(*

short summary
=================
This class provides assert statements for unsigned integers  (``UINT``)
It implements the interface :ref:`IUintAssertions`

.. <legal notes>

legal notes
=================
| SPDX-FileCopyrightText: © 2022 ekvip automation GmbH <info@ekvip.de>
| SPDX-License-Identifier: Apache-2.0
| For details check: Apache-2.0_

.. _Apache-2.0: https://www.apache.org/licenses/LICENSE-2.0

.. </legal notes>

methods and properties
=======================

*)

{attribute 'reflection'}
FUNCTION_BLOCK INTERNAL UintAssertions EXTENDS AbstactAssertion IMPLEMENTS IUintAssertions
VAR
END_VAR

(*

short summary
=================
This abstract property returns the class name of the concrete object, 
It's for debugging purpose

.. <legal notes>

legal notes
=================
| SPDX-FileCopyrightText: © 2022 ekvip automation GmbH <info@ekvip.de>
| SPDX-License-Identifier: Apache-2.0
| For details check: Apache-2.0_

.. _Apache-2.0: https://www.apache.org/licenses/LICENSE-2.0

.. </legal notes>

*)

PROPERTY className :CNM_AbstractObject.ClassName
GET
className := 'CNM_AssertionInterfaceLib.UintAssertions';
END_GET
END_PROPERTY

(*

short summary
=================
This assertion method checks if the current value is equal to the expected value

.. <legal notes>

legal notes
=================
| SPDX-FileCopyrightText: © 2022 ekvip automation GmbH <info@ekvip.de>
| SPDX-License-Identifier: Apache-2.0
| For details check: Apache-2.0_

.. _Apache-2.0: https://www.apache.org/licenses/LICENSE-2.0

.. </legal notes>

parameters
=================

*)

METHOD valueIsEqualTo
VAR_INPUT
	(* current value to check *)
	currentValue	:UINT;
	(* expected value to compare *)
	expectedValue	:UINT;
	(* message if the assertion is false *)
	message			:AssertMessage;
END_VAR
IF (currentValue <> expectedValue) THEN
	THIS^.assertionWasWrong(message, THIS^.getDebugInfo('valueIsEqualTo'));
END_IF
END_METHOD

(*

short summary
=================
This assertion method checks if the current value is even

.. <legal notes>

legal notes
=================
| SPDX-FileCopyrightText: © 2022 ekvip automation GmbH <info@ekvip.de>
| SPDX-License-Identifier: Apache-2.0
| For details check: Apache-2.0_

.. _Apache-2.0: https://www.apache.org/licenses/LICENSE-2.0

.. </legal notes>

parameters
=================

*)

METHOD valueIsEven
VAR_INPUT
	(* current value to check *)
	currentValue	:UINT;
	(* message if the assertion is false *)
	message			:Tc2_System.T_MaxString;
END_VAR
IF ((currentValue MOD 2) <> 0) THEN
	THIS^.assertionWasWrong(message, THIS^.getDebugInfo('valueIsEven'));
END_IF
END_METHOD

(*

short summary
=================
This assertion method checks if the current value is greater than the less value

.. <legal notes>

legal notes
=================
| SPDX-FileCopyrightText: © 2022 ekvip automation GmbH <info@ekvip.de>
| SPDX-License-Identifier: Apache-2.0
| For details check: Apache-2.0_

.. _Apache-2.0: https://www.apache.org/licenses/LICENSE-2.0

.. </legal notes>

parameters
=================

*)

METHOD valueIsGreaterThan
VAR_INPUT
	(* current value to check *)
	currentValue	:UINT;
	(* less than lower limit *)
	lessValue		:UINT;
	(* message if the assertion is false *)
	message			:AssertMessage;
END_VAR
IF (currentValue <= lessValue) THEN
	THIS^.assertionWasWrong(message, THIS^.getDebugInfo('valueIsGreaterThan'));
END_IF
END_METHOD

(*

short summary
=================
This assertion method checks if the current value is inside a limit

.. attention:: 
	limits are included: ``valueIsInRangeOf(3, 3, 3)`` is a true assertion

.. <legal notes>

legal notes
=================
| SPDX-FileCopyrightText: © 2022 ekvip automation GmbH <info@ekvip.de>
| SPDX-License-Identifier: Apache-2.0
| For details check: Apache-2.0_

.. _Apache-2.0: https://www.apache.org/licenses/LICENSE-2.0

.. </legal notes>

parameters
=================

*)

METHOD valueIsInRangeOf
VAR_INPUT
	(* lower limit for the current value *)
	lowerLimit		:UINT;
	(* current value to check *)
	currentValue	:UINT;
	(* upper limit for the current value *)
	upperLimit		:UINT;
	(* message if the assertion is false *)
	message			:AssertMessage;
END_VAR
IF (
	(currentValue < lowerLimit)
	OR (currentValue > upperLimit)
) THEN
	THIS^.assertionWasWrong(message, THIS^.getDebugInfo('valueIsInRangeOf'));
END_IF
END_METHOD

(*

short summary
=================
This assertion method checks if the current value is less than the greater value

.. <legal notes>

legal notes
=================
| SPDX-FileCopyrightText: © 2022 ekvip automation GmbH <info@ekvip.de>
| SPDX-License-Identifier: Apache-2.0
| For details check: Apache-2.0_

.. _Apache-2.0: https://www.apache.org/licenses/LICENSE-2.0

.. </legal notes>

parameters
=================

*)

METHOD valueIsLessThan
VAR_INPUT
	(* current value to check *)
	currentValue	:UINT;
	(* greater than upper limit *)
	greaterValue	:UINT;
	(* message if the assertion is false *)
	message			:AssertMessage;
END_VAR
IF (currentValue >= greaterValue) THEN
	THIS^.assertionWasWrong(message, THIS^.getDebugInfo('valueIsLessThan'));
END_IF
END_METHOD

(*

short summary
=================
This assertion method checks if the current value is less than or equal to the maximum value

.. <legal notes>

legal notes
=================
| SPDX-FileCopyrightText: © 2022 ekvip automation GmbH <info@ekvip.de>
| SPDX-License-Identifier: Apache-2.0
| For details check: Apache-2.0_

.. _Apache-2.0: https://www.apache.org/licenses/LICENSE-2.0

.. </legal notes>

parameters
=================

*)

METHOD valueIsMax
VAR_INPUT
	(* current value to check *)
	currentValue	:UINT;
	(* upper limit for the current value *)
	maximumValue	:UINT;
	(* message if the assertion is false *)
	message			:AssertMessage;
END_VAR
IF (currentValue > maximumValue) THEN
	THIS^.assertionWasWrong(message, THIS^.getDebugInfo('valueIsMax'));
END_IF
END_METHOD

(*

short summary
=================
This assertion method checks if the current value is greater than or equal to the minimum value

.. <legal notes>

legal notes
=================
| SPDX-FileCopyrightText: © 2022 ekvip automation GmbH <info@ekvip.de>
| SPDX-License-Identifier: Apache-2.0
| For details check: Apache-2.0_

.. _Apache-2.0: https://www.apache.org/licenses/LICENSE-2.0

.. </legal notes>

parameters
=================

*)

METHOD valueIsMin
VAR_INPUT
	(* current value to check *)
	currentValue	:UINT;
	(* lower limit for the current value *)
	minimumValue	:UINT;
	(* message if the assertion is false *)
	message			:AssertMessage;
END_VAR
IF (currentValue < minimumValue) THEN
	THIS^.assertionWasWrong(message, THIS^.getDebugInfo('valueIsMin'));
END_IF
END_METHOD

(*

short summary
=================
This assertion method checks if the current value is not equal to the unexpected value

.. <legal notes>

legal notes
=================
| SPDX-FileCopyrightText: © 2022 ekvip automation GmbH <info@ekvip.de>
| SPDX-License-Identifier: Apache-2.0
| For details check: Apache-2.0_

.. _Apache-2.0: https://www.apache.org/licenses/LICENSE-2.0

.. </legal notes>

parameters
=================

*)

METHOD valueIsNotEqualTo
VAR_INPUT
	(* current value to check *)
	currentValue	:UINT;
	(* unexpected value to compare *)
	unexpectedValue	:UINT;
	(* message if the assertion is false *)
	message			:AssertMessage;
END_VAR
IF (currentValue = unexpectedValue) THEN
	THIS^.assertionWasWrong(message, THIS^.getDebugInfo('valueIsNotEqualTo'));
END_IF
END_METHOD

(*

short summary
=================
This assertion method checks if the current value is odd

.. <legal notes>

legal notes
=================
| SPDX-FileCopyrightText: © 2022 ekvip automation GmbH <info@ekvip.de>
| SPDX-License-Identifier: Apache-2.0
| For details check: Apache-2.0_

.. _Apache-2.0: https://www.apache.org/licenses/LICENSE-2.0

.. </legal notes>

parameters
=================

*)

METHOD valueIsOdd
VAR_INPUT
	(* current value to check *)
	currentValue	:UINT;
	(* message if the assertion is false *)
	message			:AssertMessage;
END_VAR
IF ((currentValue MOD 2) = 0) THEN
	THIS^.assertionWasWrong(message, THIS^.getDebugInfo('valueIsOdd'));
END_IF
END_METHOD

END_FUNCTION_BLOCK

(* stored: Version 1.1.0.1, ProductVersion 3.1.4024.11
   POU UintAssertions: Id {84cb69cf-f417-49b9-b9fb-83ea1eacb025}, SpecialFunc None
   Property className: Id {717aea52-1536-4993-b7ba-8e37d488112e}
   Get Get: Id {60fc7789-fc7e-4786-bf4b-497abe8d15f4}
   Method valueIsEqualTo: Id {739d9688-b3dc-4915-b83f-b86b0c2408ab}
   Method valueIsEven: Id {3172bec8-17fb-4c51-b251-19c2045cdc94}
   Method valueIsGreaterThan: Id {2b5272d3-4f84-4f55-b2bb-d81099b2fc6b}
   Method valueIsInRangeOf: Id {62b90422-dc55-4051-9a08-f27c70eb6b2a}
   Method valueIsLessThan: Id {928f728b-87ec-4678-959d-02e8c8345da7}
   Method valueIsMax: Id {cd551aba-e29b-431d-bb53-4be64bc96f3a}
   Method valueIsMin: Id {f1408381-0b8d-4460-9550-99172563b349}
   Method valueIsNotEqualTo: Id {982a51ac-59b2-479a-9951-4fe6aa93ad71}
   Method valueIsOdd: Id {23c2b606-1ecc-4533-9574-66777a7eaff2} *)
